// TIA Portal V15.1 export
// export: Created 2024-05-17T05:38:49.0670589Z, ExportSetting WithDefaults, DisplayName Totally Integrated Automation Portal, DisplayVersion V15.1 Update 5, DisplayName TIA Portal Openness, DisplayVersion V15.1 Update 5, DisplayName SINAMICS Startdrive Advanced, DisplayVersion V15.1, DisplayName G130, G150, S120, S150, SINAMICS MV, S210, DisplayVersion V15.1, DisplayName G110M, G120, G120C, G120D, G120P, DisplayVersion V15.1, DisplayName STEP 7 Professional, DisplayVersion V15.1 Update 5, DisplayName STEP 7 Safety, DisplayVersion V15.1, DisplayName WinCC Professional, DisplayVersion V15.1 Update 5, DisplayName SIMATIC Visualization Architect, DisplayVersion V15.1
FUNCTION_BLOCK "LGBExtCross2W2S-MoviFitFCPN"   // FB6653, FBD
TITLE = LGBExtCross2W2S-MoviFitFCPN
{ S7_Optimized_Access := 'TRUE' }
AUTHOR : ENGIE
FAMILY : Actuator
VERSION : 0.1
// stored: AutoNumber false, IsIECCheckEnabled false, IsRetainMemResEnabled false, MemoryReserve 100, SetENOAutomatically False, UDAEnableTagReadback false
   VAR_INPUT
      I_MotorProtection { ExternalAccessible := 'False'; ExternalVisible := 'False'; ExternalWritable := 'False'} : Bool;   // Motor protection
      I_BeltControlLeftDet { ExternalAccessible := 'False'; ExternalVisible := 'False'; ExternalWritable := 'False'} : Bool;   // Sensor Belt Control CrossConv left
      I_BeltControlRightDet { ExternalAccessible := 'False'; ExternalVisible := 'False'; ExternalWritable := 'False'} : Bool;   // Sensor Belt Control CrossConv right
      I_AlarmResetPB { ExternalAccessible := 'False'; ExternalVisible := 'False'; ExternalWritable := 'False'} : Bool;   // Alarm Reset Pushbutton is Activated
      I_SafetyStatusWord { ExternalAccessible := 'False'; ExternalVisible := 'False'; ExternalWritable := 'False'} : Word;   // Safety status word
      I_SafetyControlWord { ExternalAccessible := 'False'; ExternalVisible := 'False'; ExternalWritable := 'False'} : Word;   // Safety control word
      I_SafetyOk { ExternalAccessible := 'False'; ExternalVisible := 'False'; ExternalWritable := 'False'} : Bool;   // Safety ok
      I_MotionStopOk { ExternalAccessible := 'False'; ExternalVisible := 'False'; ExternalWritable := 'False'} : Bool;   // Safety Ok / The motion stop is Ok
      I_LSpdSetMotorCmd { ExternalAccessible := 'False'; ExternalVisible := 'False'; ExternalWritable := 'False'} : Bool;   // Low speed Set Command from function after interlock
      I_HSpdSetMotorCmd { ExternalAccessible := 'False'; ExternalVisible := 'False'; ExternalWritable := 'False'} : Bool;   // High Speed Set Command from function after Interlock
      I_LSpdResMotorCmd { ExternalAccessible := 'False'; ExternalVisible := 'False'; ExternalWritable := 'False'} : Bool;   // Low speed Reset Command from function after interlock
      I_HSpdResMotorCmd { ExternalAccessible := 'False'; ExternalVisible := 'False'; ExternalWritable := 'False'} : Bool;   // High speed Reset Command from function after Interlock
      I_LowSpeed { ExternalAccessible := 'False'; ExternalVisible := 'False'; ExternalWritable := 'False'} : Real;   // Low speed value 0-100%
      I_HighSpeed { ExternalAccessible := 'False'; ExternalVisible := 'False'; ExternalWritable := 'False'} : Real;   // High speed value 0-100%
      I_ReleaseBrake { ExternalAccessible := 'False'; ExternalVisible := 'False'; ExternalWritable := 'False'} : Bool;   // Release brake
   END_VAR
   VAR_OUTPUT
      O_ReleaseBrake { ExternalAccessible := 'False'; ExternalVisible := 'False'; ExternalWritable := 'False'} : Bool;   // Release the brake of the Motor
      O_Active { ExternalAccessible := 'False'; ExternalVisible := 'False'; ExternalWritable := 'False'} : Bool;   // Motor loop Active
      O_AlarmABCondition { ExternalAccessible := 'False'; ExternalVisible := 'False'; ExternalWritable := 'False'} : Bool;   // Alarm AB Condition
      O_AlarmA { ExternalAccessible := 'False'; ExternalVisible := 'False'; ExternalWritable := 'False'} : Bool;   // Alarm A
      O_AlarmB { ExternalAccessible := 'False'; ExternalVisible := 'False'; ExternalWritable := 'False'} : Bool;   // Alarm B
      O_AlarmC { ExternalAccessible := 'False'; ExternalVisible := 'False'; ExternalWritable := 'False'} : Bool;   // Alarm C
      O_AlarmD { ExternalAccessible := 'False'; ExternalVisible := 'False'; ExternalWritable := 'False'} : Bool;   // Alarm D
      H_AlarmDWord { ExternalAccessible := 'False'; ExternalVisible := 'False'; ExternalWritable := 'False'} : DWord;   // Alarm Word
   END_VAR
   VAR_IN_OUT
      IO_Modes : "Modes";   // Modes
      H_HMI : "H_HMI";
      "H_GBExtCross2W2S-MoviFitFCPN" : "H_GBExtCross2W2S-MoviFitFCPN";   // HMI UDT
      C_Config : "ExtCrossConfig";   // Config
   END_VAR
   VAR
      AA_MotorProtector { ExternalAccessible := 'False'; ExternalVisible := 'False'; ExternalWritable := 'False'} : Bool;   // Motorprotection Tripped / Motor Protection Tripped
      AA_SafetySwitch { ExternalAccessible := 'False'; ExternalVisible := 'False'; ExternalWritable := 'False'} : Bool;   // Safety Switch Not Ok
      AA_NoBusControl { ExternalAccessible := 'False'; ExternalVisible := 'False'; ExternalWritable := 'False'} : Bool;   // Bus control inactive
      AB_STO { ExternalAccessible := 'False'; ExternalVisible := 'False'; ExternalWritable := 'False'} : Bool;   // Safety Switch Not Ok / Safety output to drive is active but no response from drive that the safety is ok (STO)
      AB_BeltControlLeftDet { ExternalAccessible := 'False'; ExternalVisible := 'False'; ExternalWritable := 'False'} : Bool;   // Belt Check Cross Conveyor Left Side
      AB_BeltControlRightDet { ExternalAccessible := 'False'; ExternalVisible := 'False'; ExternalWritable := 'False'} : Bool;   // Belt Check Cross Conveyor Right Side
      AB_Alarm { ExternalAccessible := 'False'; ExternalVisible := 'False'; ExternalWritable := 'False'} : Bool;   // Frequency Control
      AD_Warning { ExternalAccessible := 'False'; ExternalVisible := 'False'; ExternalWritable := 'False'} : Bool;   // Frequency Control
      AD_MotionStop { ExternalAccessible := 'False'; ExternalVisible := 'False'; ExternalWritable := 'False'} : Bool;   // Motion Stop
      SafetyOk { ExternalAccessible := 'False'; ExternalVisible := 'False'; ExternalWritable := 'False'} : Bool;   // Safety Ok
      ParameterSet { ExternalAccessible := 'False'; ExternalVisible := 'False'; ExternalWritable := 'False'} : Bool;   // Active parameter set
      SetFrequency { ExternalAccessible := 'False'; ExternalVisible := 'False'; ExternalWritable := 'False'} : Real;   // Set frequency dependant on config
      ResFrequency { ExternalAccessible := 'False'; ExternalVisible := 'False'; ExternalWritable := 'False'} : Real;   // Reset frequency dependant on config
      MotorProtectionAlarmABCond { ExternalAccessible := 'False'; ExternalVisible := 'False'; ExternalWritable := 'False'} : Bool;   // Motor protection alarm condition
      SafetySwitchAlarmABCond { ExternalAccessible := 'False'; ExternalVisible := 'False'; ExternalWritable := 'False'} : Bool;   // Safety Switch alarm condition
      DriveFaultAlarm { ExternalAccessible := 'False'; ExternalVisible := 'False'; ExternalWritable := 'False'} : Bool;   // Drive fault alarm
      DriveFaultAlarmABCond { ExternalAccessible := 'False'; ExternalVisible := 'False'; ExternalWritable := 'False'} : Bool;   // Drive fault alarm condition
      STOAlarmABCond { ExternalAccessible := 'False'; ExternalVisible := 'False'; ExternalWritable := 'False'} : Bool;   // Drive fault alarm condition / STO feedback fault alarm condition
      EnableAlarmHWSR { ExternalAccessible := 'False'; ExternalVisible := 'False'; ExternalWritable := 'False'} : Bool;   // Enable Alarms from the hardware
      EnableAlarmHW { ExternalAccessible := 'False'; ExternalVisible := 'False'; ExternalWritable := 'False'} : Bool;   // Enable Alarms from the hardware
      Start { ExternalAccessible := 'False'; ExternalVisible := 'False'; ExternalWritable := 'False'} : Bool;   // Start command to drive
      SetpointSpeed { ExternalAccessible := 'False'; ExternalVisible := 'False'; ExternalWritable := 'False'} : Real;   // Setpoint speed
      SetpointSpeedCalc { ExternalAccessible := 'False'; ExternalVisible := 'False'; ExternalWritable := 'False'} : Real;   // Setpoint speed to drive / Setpoint speed
      OutputStageEnabled { ExternalAccessible := 'False'; ExternalVisible := 'False'; ExternalWritable := 'False'} : Bool;   // Inverter output stage is enabled
      MaintenanceSwitch { ExternalAccessible := 'False'; ExternalVisible := 'False'; ExternalWritable := 'False'} : Bool;   // Maintenance switch activated (1=mains OFF)
      PODataEnabled { ExternalAccessible := 'False'; ExternalVisible := 'False'; ExternalWritable := 'False'} : Bool;   // Process data is enabled (1 = Drive can be controlled via fieldbus)
      PODataDisabled { ExternalAccessible := 'False'; ExternalVisible := 'False'; ExternalWritable := 'False'} : Bool;   // Process data is enabled (1 = Drive can be controlled via fieldbus)
      Fault { ExternalAccessible := 'False'; ExternalVisible := 'False'; ExternalWritable := 'False'} : Bool;   // Fault present
      Brake { ExternalAccessible := 'False'; ExternalVisible := 'False'; ExternalWritable := 'False'} : Bool;   // Brake status
      ActorVoltageOverloadDO00 { ExternalAccessible := 'False'; ExternalVisible := 'False'; ExternalWritable := 'False'} : Bool;   // Short circuit / overload of the actuator voltage for digital output DO00
      ActorVoltageOverloadDO01 { ExternalAccessible := 'False'; ExternalVisible := 'False'; ExternalWritable := 'False'} : Bool;   // Short circuit / overload of the actuator voltage for digital output DO01
      ActorVoltageOverloadDO02 { ExternalAccessible := 'False'; ExternalVisible := 'False'; ExternalWritable := 'False'} : Bool;   // Short circuit / overload of the actuator voltage for digital output DO02
      ActorVoltageOverloadDO03 { ExternalAccessible := 'False'; ExternalVisible := 'False'; ExternalWritable := 'False'} : Bool;   // Short circuit / overload of the actuator voltage for digital output DO03
      SensorVoltageOverloadGroup1 { ExternalAccessible := 'False'; ExternalVisible := 'False'; ExternalWritable := 'False'} : Bool;   // Short circuit / overload of the sensor suuply group 1 (VO24-I)
      SensorVoltageOverloadGroup2 { ExternalAccessible := 'False'; ExternalVisible := 'False'; ExternalWritable := 'False'} : Bool;   // Short circuit / overload of the sensor suuply group 2 (VO24-I)
      SensorVoltageOverloadGroup3 { ExternalAccessible := 'False'; ExternalVisible := 'False'; ExternalWritable := 'False'} : Bool;   // Short circuit / overload of the sensor suuply group 3 (VO24-I)
      SensorVoltageOverloadGroup4 { ExternalAccessible := 'False'; ExternalVisible := 'False'; ExternalWritable := 'False'} : Bool;   // Short circuit / overload of the sensor suuply group 4 (VO24-I)
      "Undervoltage24V-S" { ExternalAccessible := 'False'; ExternalVisible := 'False'; ExternalWritable := 'False'} : Bool;   // Value falls below the power limit for the actuator voltage DO00-03
      "InverterVoltageNotApplied24V-P" { ExternalAccessible := 'False'; ExternalVisible := 'False'; ExternalWritable := 'False'} : Bool;   // Presence of 24V_P for integrated inverter (FC) or external MOVIMOT (1=24V_P not present)
      MOVIFITSystemFault { ExternalAccessible := 'False'; ExternalVisible := 'False'; ExternalWritable := 'False'} : Bool;   // MOVIFIT system fault
      DriveReady { ExternalAccessible := 'False'; ExternalVisible := 'False'; ExternalWritable := 'False'} : Bool;   // Motor Loop Active / Drive ready
      BeltControlLeftAlarmABCondition { ExternalAccessible := 'False'; ExternalVisible := 'False'; ExternalWritable := 'False'} : Bool;   // Belt Control AB Condition
      BeltControlRightAlarmABCondition { ExternalAccessible := 'False'; ExternalVisible := 'False'; ExternalWritable := 'False'} : Bool;   // Belt Control AB Condition
      BeltPulseCountLeft { ExternalAccessible := 'False'; ExternalVisible := 'False'; ExternalWritable := 'False'} : DInt;   // Temp
      BeltPulseCountRight { ExternalAccessible := 'False'; ExternalVisible := 'False'; ExternalWritable := 'False'} : DInt;   // Temp
      BeltPosEdgeLeft1 { ExternalAccessible := 'False'; ExternalVisible := 'False'; ExternalWritable := 'False'} : Bool;   // Pos Edge
      BeltPosEdgeLeft2 { ExternalAccessible := 'False'; ExternalVisible := 'False'; ExternalWritable := 'False'} : Bool;   // Pos Edge
      BeltPosEdgeRight1 { ExternalAccessible := 'False'; ExternalVisible := 'False'; ExternalWritable := 'False'} : Bool;   // Pos Edge
      BeltPosEdgeRight2 { ExternalAccessible := 'False'; ExternalVisible := 'False'; ExternalWritable := 'False'} : Bool;   // Pos Edge
      InitBeltCounterLeft { ExternalAccessible := 'False'; ExternalVisible := 'False'; ExternalWritable := 'False'} : Bool;   // Init
      InitBeltCounterRight { ExternalAccessible := 'False'; ExternalVisible := 'False'; ExternalWritable := 'False'} : Bool;   // Init
      AlarmA { ExternalAccessible := 'False'; ExternalVisible := 'False'; ExternalWritable := 'False'} : Bool;   // Alarm A
      AlarmB { ExternalAccessible := 'False'; ExternalVisible := 'False'; ExternalWritable := 'False'} : Bool;   // Alarm B
      AlarmC { ExternalAccessible := 'False'; ExternalVisible := 'False'; ExternalWritable := 'False'} : Bool;   // Alarm C
      AlarmD { ExternalAccessible := 'False'; ExternalVisible := 'False'; ExternalWritable := 'False'} : Bool;   // Alarm D
      Ramp { ExternalAccessible := 'False'; ExternalVisible := 'False'; ExternalWritable := 'False'} : DInt;   // Ramp
      RampToDrive { ExternalAccessible := 'False'; ExternalVisible := 'False'; ExternalWritable := 'False'} : Time;   // Calculated Ramp send in miliseconds
      _BeltControlRight { ExternalAccessible := 'False'; ExternalVisible := 'False'; ExternalWritable := 'False'} : "L1AlarmMultiIn";   // FB
      _BeltControlLeft { ExternalAccessible := 'False'; ExternalVisible := 'False'; ExternalWritable := 'False'} : "L1AlarmMultiIn";   // FB
      _InitBeltCntLeft { ExternalAccessible := 'False'; ExternalVisible := 'False'; ExternalWritable := 'False'} : "LChangeOfState";   // FB
      _InitBeltCntRight { ExternalAccessible := 'False'; ExternalVisible := 'False'; ExternalWritable := 'False'} : "LChangeOfState";   // FB
      _MoviFitPN { ExternalAccessible := 'False'; ExternalVisible := 'False'; ExternalWritable := 'False'} : "LGBSEW-MoviFitFCPN";   // FB / SEW MOVIFIT FC
      _MotorProtection { ExternalAccessible := 'False'; ExternalVisible := 'False'; ExternalWritable := 'False'} : "L1AlarmMultiIn";   // FB
      _SafetySwitch { ExternalAccessible := 'False'; ExternalVisible := 'False'; ExternalWritable := 'False'} : "L1AlarmMultiIn";   // FB
      _DriveFault { ExternalAccessible := 'False'; ExternalVisible := 'False'; ExternalWritable := 'False'} : "L1AlarmMultiIn";   // FB
      _STO { ExternalAccessible := 'False'; ExternalVisible := 'False'; ExternalWritable := 'False'} : "L1AlarmMultiIn";   // FB
      _MotionStop { ExternalAccessible := 'False'; ExternalVisible := 'False'; ExternalWritable := 'False'} : "L1AlarmMultiIn";   // FB
      T_STOAlarm { ExternalAccessible := 'False'; ExternalVisible := 'False'; ExternalWritable := 'False'} : TON_TIME;   // Timer
      T_Reboot { ExternalAccessible := 'False'; ExternalVisible := 'False'; ExternalWritable := 'False'} : TON_TIME;   // Timer
   END_VAR
   VAR_TEMP   // added for the SCL form of the ladder/FBD networks
      _w1 : Bool;
      _w2 : Bool;
      _w3 : Bool;
      _w4 : Bool;
   END_VAR
BEGIN

NETWORK
TITLE = **** 1 - Inputs **** Init Belt Control Set And Reset Direction
// Init Belt Control Set And Reset Direction
      CALL  #_InitBeltCntLeft
      ( I_In     := #I_BeltControlLeftDet,
        O_OutPut := #InitBeltCounterLeft
      );
      NOP   0;

      CALL  #_InitBeltCntRight
      ( I_In     := #I_BeltControlRightDet,
        O_OutPut := #InitBeltCounterRight
      );
      NOP   0;

      A(;
      O     #InitBeltCounterLeft;
      O;
      A     #IO_Modes.LMode.ManualMode;
      A     #IO_Modes.LMode.AlarmResetPB;
      );
      JCN   NCSet;
      L     0;
      T     #BeltPulseCountLeft;
NCSet:NOP   0;

      A(;
      O     #InitBeltCounterRight;
      O;
      A     #IO_Modes.LMode.ManualMode;
      A     #IO_Modes.LMode.AlarmResetPB;
      );
      JCN   NCReset;
      L     0;
      T     #BeltPulseCountRight;
NCReset:NOP   0;


REGION Network 2: **** 1 - Inputs **** Safety Ok
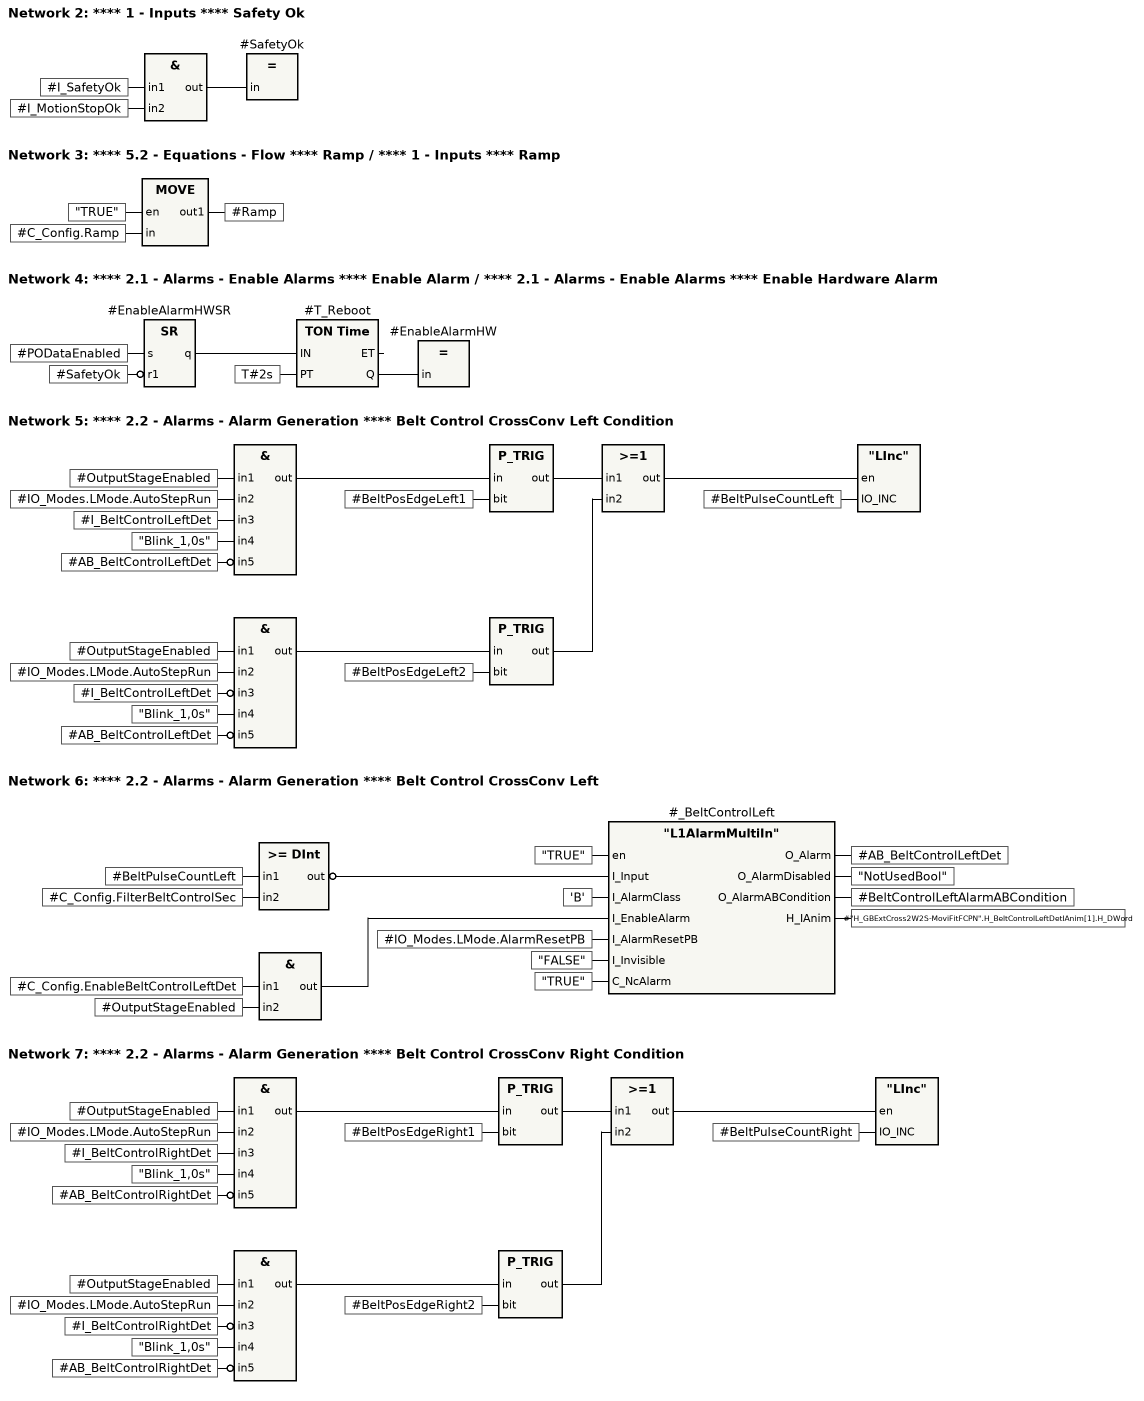
   #SafetyOk := #I_SafetyOk AND #I_MotionStopOk;
END_REGION

REGION Network 3: **** 5.2 - Equations - Flow **** Ramp / **** 1 - Inputs **** Ramp
   IF "TRUE" THEN #Ramp := #C_Config.Ramp; END_IF;
END_REGION

REGION Network 4: **** 2.1 - Alarms - Enable Alarms **** Enable Alarm / **** 2.1 - Alarms - Enable Alarms **** Enable Hardware Alarm
   // Enable Alarm / Enable Hardware Alarm
   IF #PODataEnabled THEN
       #EnableAlarmHWSR := TRUE;   // SR flip-flop
   END_IF;
   IF NOT #SafetyOk THEN #EnableAlarmHWSR := FALSE; END_IF;
   #T_Reboot(IN := #EnableAlarmHWSR, PT := T#2s);   // TON
   #EnableAlarmHW := #T_Reboot.Q;
END_REGION

REGION Network 5: **** 2.2 - Alarms - Alarm Generation **** Belt Control CrossConv Left Condition
   // Belt Control CrossConv Set Condition
   #_w1 := #OutputStageEnabled AND #IO_Modes.LMode.AutoStepRun AND #I_BeltControlLeftDet AND "Blink_1,0s" AND NOT #AB_BeltControlLeftDet;
   #_w2 := #_w1 AND NOT #BeltPosEdgeLeft1;   // rising edge
   #BeltPosEdgeLeft1 := #_w1;
   #_w3 := #OutputStageEnabled AND #IO_Modes.LMode.AutoStepRun AND NOT #I_BeltControlLeftDet AND "Blink_1,0s" AND NOT #AB_BeltControlLeftDet;
   #_w4 := #_w3 AND NOT #BeltPosEdgeLeft2;   // rising edge
   #BeltPosEdgeLeft2 := #_w3;
   IF #_w2 OR #_w4 THEN "LInc"(IO_INC := #BeltPulseCountLeft); END_IF;
END_REGION

REGION Network 6: **** 2.2 - Alarms - Alarm Generation **** Belt Control CrossConv Left
   // Belt Control CrossConv Set
   IF "TRUE" THEN
       #_BeltControlLeft(I_Input := NOT (#BeltPulseCountLeft >= #C_Config.FilterBeltControlSec),   // "L1AlarmMultiIn"
                         I_AlarmClass := 'B',
                         I_EnableAlarm := #C_Config.EnableBeltControlLeftDet AND #OutputStageEnabled,
                         I_AlarmResetPB := #IO_Modes.LMode.AlarmResetPB,
                         I_Invisible := "FALSE",
                         C_NcAlarm := "TRUE",
                         O_Alarm => #AB_BeltControlLeftDet,
                         O_AlarmDisabled => "NotUsedBool",
                         O_AlarmABCondition => #BeltControlLeftAlarmABCondition,
                         H_IAnim => #"H_GBExtCross2W2S-MoviFitFCPN".H_BeltControlLeftDetIAnim[1].H_DWord);
   END_IF;
END_REGION

REGION Network 7: **** 2.2 - Alarms - Alarm Generation **** Belt Control CrossConv Right Condition
   // Belt Control CrossConv Set Condition
   #_w1 := #OutputStageEnabled AND #IO_Modes.LMode.AutoStepRun AND #I_BeltControlRightDet AND "Blink_1,0s" AND NOT #AB_BeltControlRightDet;
   #_w2 := #_w1 AND NOT #BeltPosEdgeRight1;   // rising edge
   #BeltPosEdgeRight1 := #_w1;
   #_w3 := #OutputStageEnabled AND #IO_Modes.LMode.AutoStepRun AND NOT #I_BeltControlRightDet AND "Blink_1,0s" AND NOT #AB_BeltControlRightDet;
   #_w4 := #_w3 AND NOT #BeltPosEdgeRight2;   // rising edge
   #BeltPosEdgeRight2 := #_w3;
   IF #_w2 OR #_w4 THEN "LInc"(IO_INC := #BeltPulseCountRight); END_IF;
END_REGION

REGION Network 8: **** 2.2 - Alarms - Alarm Generation **** Belt Control CrossConv Right
   // Belt Control CrossConv Set
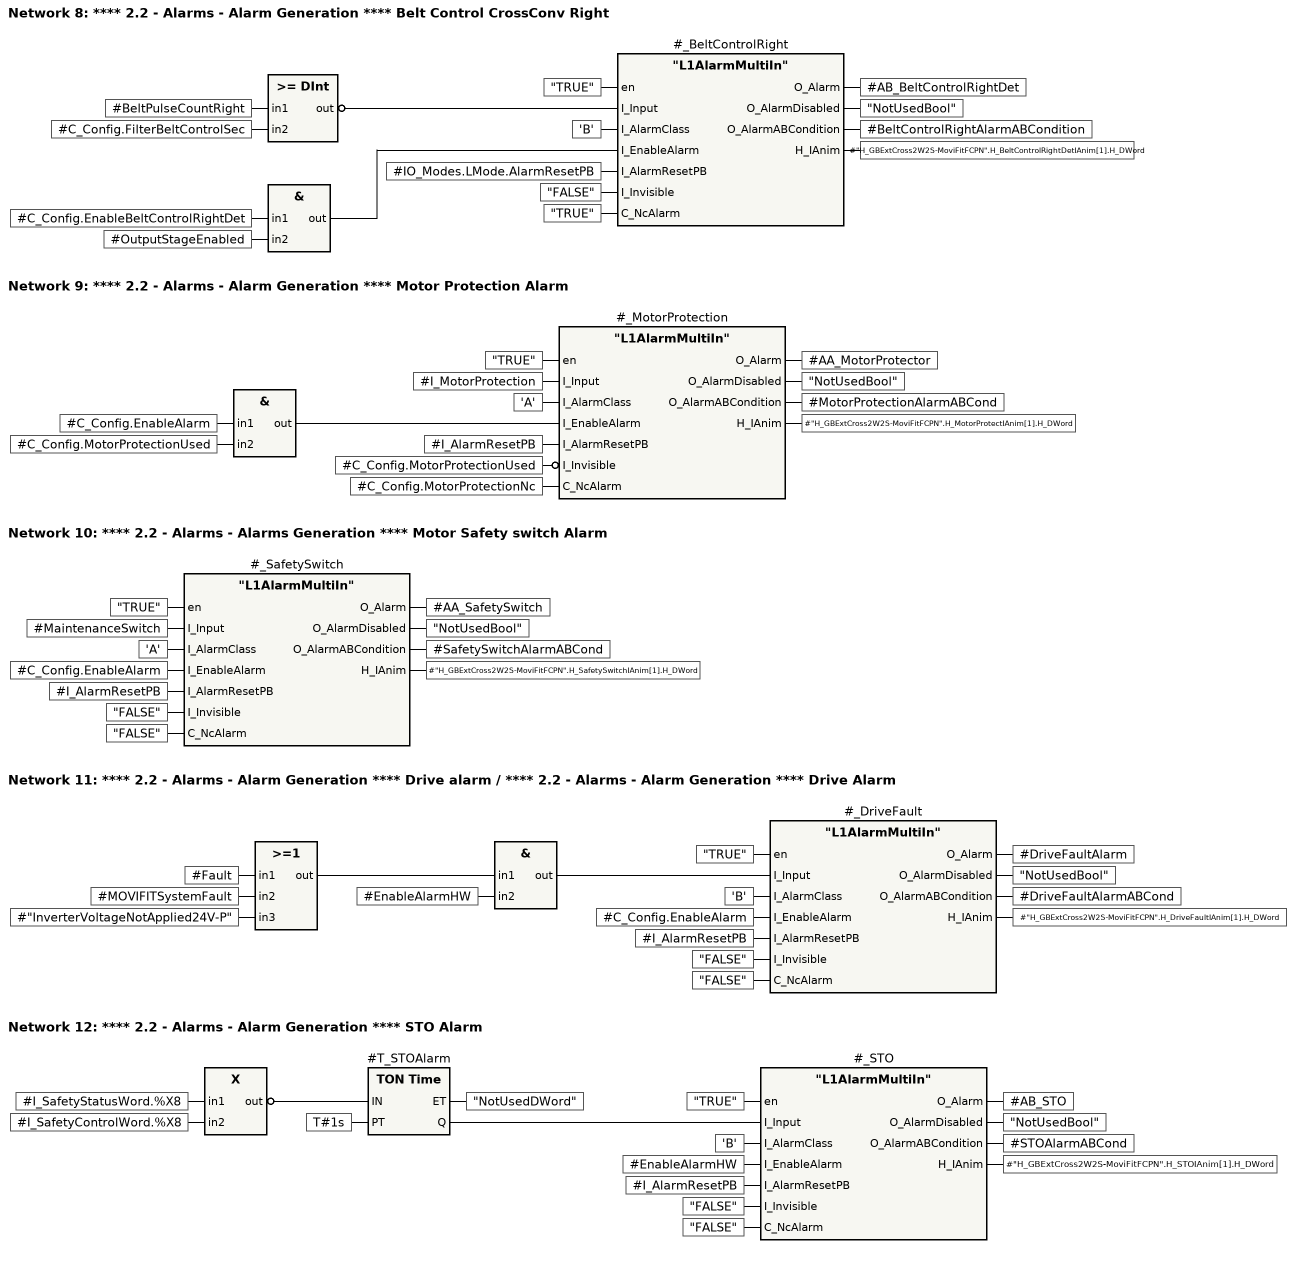
   IF "TRUE" THEN
       #_BeltControlRight(I_Input := NOT (#BeltPulseCountRight >= #C_Config.FilterBeltControlSec),   // "L1AlarmMultiIn"
                          I_AlarmClass := 'B',
                          I_EnableAlarm := #C_Config.EnableBeltControlRightDet AND #OutputStageEnabled,
                          I_AlarmResetPB := #IO_Modes.LMode.AlarmResetPB,
                          I_Invisible := "FALSE",
                          C_NcAlarm := "TRUE",
                          O_Alarm => #AB_BeltControlRightDet,
                          O_AlarmDisabled => "NotUsedBool",
                          O_AlarmABCondition => #BeltControlRightAlarmABCondition,
                          H_IAnim => #"H_GBExtCross2W2S-MoviFitFCPN".H_BeltControlRightDetIAnim[1].H_DWord);
   END_IF;
END_REGION

REGION Network 9: **** 2.2 - Alarms - Alarm Generation **** Motor Protection Alarm
   // Motor Protection Alarm
   IF "TRUE" THEN
       #_MotorProtection(I_Input := #I_MotorProtection,   // "L1AlarmMultiIn"
                         I_AlarmClass := 'A',
                         I_EnableAlarm := #C_Config.EnableAlarm AND #C_Config.MotorProtectionUsed,
                         I_AlarmResetPB := #I_AlarmResetPB,
                         I_Invisible := NOT #C_Config.MotorProtectionUsed,
                         C_NcAlarm := #C_Config.MotorProtectionNc,
                         O_Alarm => #AA_MotorProtector,
                         O_AlarmDisabled => "NotUsedBool",
                         O_AlarmABCondition => #MotorProtectionAlarmABCond,
                         H_IAnim => #"H_GBExtCross2W2S-MoviFitFCPN".H_MotorProtectIAnim[1].H_DWord);
   END_IF;
END_REGION

REGION Network 10: **** 2.2 - Alarms - Alarms Generation **** Motor Safety switch Alarm
   // Motor Safety switch Alarm
   IF "TRUE" THEN
       #_SafetySwitch(I_Input := #MaintenanceSwitch,   // "L1AlarmMultiIn"
                      I_AlarmClass := 'A',
                      I_EnableAlarm := #C_Config.EnableAlarm,
                      I_AlarmResetPB := #I_AlarmResetPB,
                      I_Invisible := "FALSE",
                      C_NcAlarm := "FALSE",
                      O_Alarm => #AA_SafetySwitch,
                      O_AlarmDisabled => "NotUsedBool",
                      O_AlarmABCondition => #SafetySwitchAlarmABCond,
                      H_IAnim => #"H_GBExtCross2W2S-MoviFitFCPN".H_SafetySwitchIAnim[1].H_DWord);
   END_IF;
END_REGION

REGION Network 11: **** 2.2 - Alarms - Alarm Generation **** Drive alarm / **** 2.2 - Alarms - Alarm Generation **** Drive Alarm
   IF "TRUE" THEN
       #_DriveFault(I_Input := (#Fault OR #MOVIFITSystemFault OR #"InverterVoltageNotApplied24V-P") AND #EnableAlarmHW,   // "L1AlarmMultiIn"
                    I_AlarmClass := 'B',
                    I_EnableAlarm := #C_Config.EnableAlarm,
                    I_AlarmResetPB := #I_AlarmResetPB,
                    I_Invisible := "FALSE",
                    C_NcAlarm := "FALSE",
                    O_Alarm => #DriveFaultAlarm,
                    O_AlarmDisabled => "NotUsedBool",
                    O_AlarmABCondition => #DriveFaultAlarmABCond,
                    H_IAnim => #"H_GBExtCross2W2S-MoviFitFCPN".H_DriveFaultIAnim[1].H_DWord);
   END_IF;
END_REGION

REGION Network 12: **** 2.2 - Alarms - Alarm Generation **** STO Alarm
   #T_STOAlarm(IN := NOT (#I_SafetyStatusWord.%X8 XOR #I_SafetyControlWord.%X8),   // TON
               PT := T#1s,
               ET => "NotUsedDWord");
   IF "TRUE" THEN
       #_STO(I_Input := #T_STOAlarm.Q,   // "L1AlarmMultiIn"
             I_AlarmClass := 'B',
             I_EnableAlarm := #EnableAlarmHW,
             I_AlarmResetPB := #I_AlarmResetPB,
             I_Invisible := "FALSE",
             C_NcAlarm := "FALSE",
             O_Alarm => #AB_STO,
             O_AlarmDisabled => "NotUsedBool",
             O_AlarmABCondition => #STOAlarmABCond,
             H_IAnim => #"H_GBExtCross2W2S-MoviFitFCPN".H_STOIAnim[1].H_DWord);
   END_IF;
END_REGION

REGION Network 13: **** 2.2 - Alarms - Alarm Generation **** MotionStop Warning
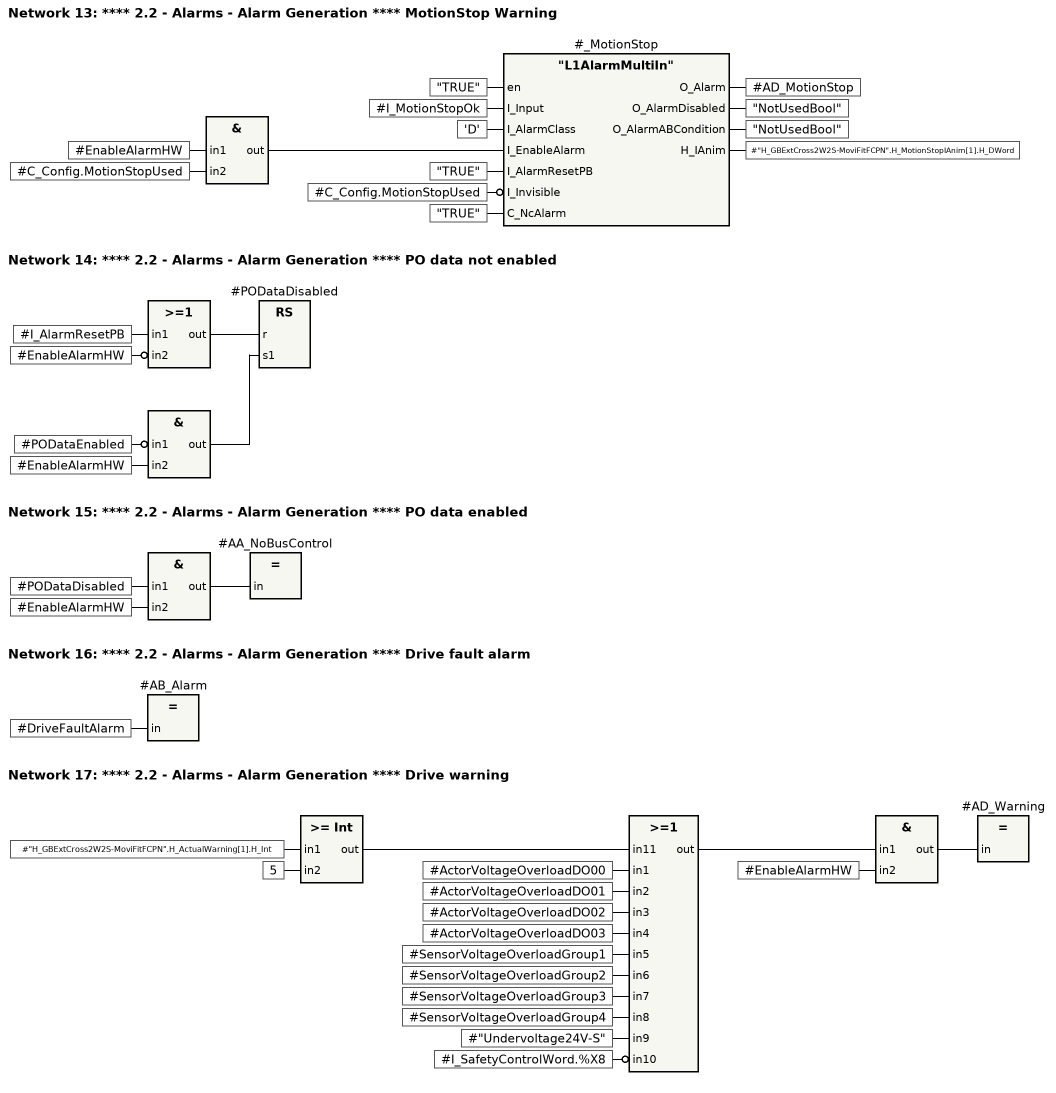
   IF "TRUE" THEN
       #_MotionStop(I_Input := #I_MotionStopOk,   // "L1AlarmMultiIn"
                    I_AlarmClass := 'D',
                    I_EnableAlarm := #EnableAlarmHW AND #C_Config.MotionStopUsed,
                    I_AlarmResetPB := "TRUE",
                    I_Invisible := NOT #C_Config.MotionStopUsed,
                    C_NcAlarm := "TRUE",
                    O_Alarm => #AD_MotionStop,
                    O_AlarmDisabled => "NotUsedBool",
                    O_AlarmABCondition => "NotUsedBool",
                    H_IAnim => #"H_GBExtCross2W2S-MoviFitFCPN".H_MotionStopIAnim[1].H_DWord);
   END_IF;
END_REGION

REGION Network 14: **** 2.2 - Alarms - Alarm Generation **** PO data not enabled
   IF #I_AlarmResetPB OR NOT #EnableAlarmHW THEN
       #PODataDisabled := FALSE;   // RS flip-flop
   END_IF;
   IF NOT #PODataEnabled AND #EnableAlarmHW THEN #PODataDisabled := TRUE; END_IF;
END_REGION

REGION Network 15: **** 2.2 - Alarms - Alarm Generation **** PO data enabled
   #AA_NoBusControl := #PODataDisabled AND #EnableAlarmHW;
END_REGION

REGION Network 16: **** 2.2 - Alarms - Alarm Generation **** Drive fault alarm
   // Drive fault
   #AB_Alarm := #DriveFaultAlarm;
END_REGION

REGION Network 17: **** 2.2 - Alarms - Alarm Generation **** Drive warning
   #AD_Warning := ((#"H_GBExtCross2W2S-MoviFitFCPN".H_ActualWarning[1].H_Int >= 5) OR #ActorVoltageOverloadDO00 OR #ActorVoltageOverloadDO01 OR #ActorVoltageOverloadDO02 OR #ActorVoltageOverloadDO03 OR #SensorVoltageOverloadGroup1 OR #SensorVoltageOverloadGroup2 OR #SensorVoltageOverloadGroup3 OR #SensorVoltageOverloadGroup4 OR #"Undervoltage24V-S" OR NOT #I_SafetyControlWord.%X8) AND #EnableAlarmHW;
END_REGION

REGION Network 18: **** 4.6 - Machine Status - Indication **** Icon Animation
   // Icon Animation
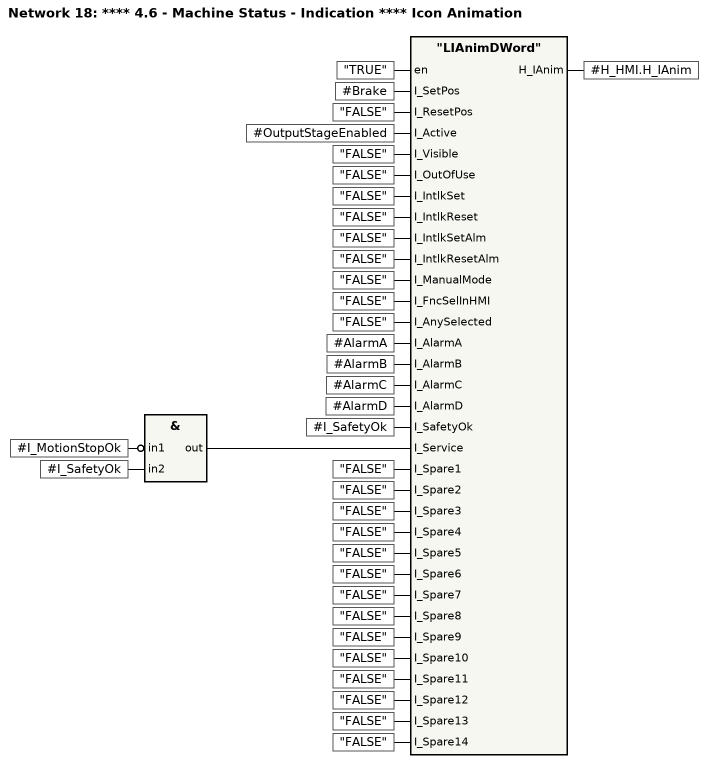
   IF "TRUE" THEN
       "LIAnimDWord"(I_SetPos := #Brake,
                     I_ResetPos := "FALSE",
                     I_Active := #OutputStageEnabled,
                     I_Visible := "FALSE",
                     I_OutOfUse := "FALSE",
                     I_IntlkSet := "FALSE",
                     I_IntlkReset := "FALSE",
                     I_IntlkSetAlm := "FALSE",
                     I_IntlkResetAlm := "FALSE",
                     I_ManualMode := "FALSE",
                     I_FncSelInHMI := "FALSE",
                     I_AnySelected := "FALSE",
                     I_AlarmA := #AlarmA,
                     I_AlarmB := #AlarmB,
                     I_AlarmC := #AlarmC,
                     I_AlarmD := #AlarmD,
                     I_SafetyOk := #I_SafetyOk,
                     I_Service := NOT #I_MotionStopOk AND #I_SafetyOk,
                     I_Spare1 := "FALSE",
                     I_Spare2 := "FALSE",
                     I_Spare3 := "FALSE",
                     I_Spare4 := "FALSE",
                     I_Spare5 := "FALSE",
                     I_Spare6 := "FALSE",
                     I_Spare7 := "FALSE",
                     I_Spare8 := "FALSE",
                     I_Spare9 := "FALSE",
                     I_Spare10 := "FALSE",
                     I_Spare11 := "FALSE",
                     I_Spare12 := "FALSE",
                     I_Spare13 := "FALSE",
                     I_Spare14 := "FALSE",
                     H_IAnim => #H_HMI.H_IAnim);
   END_IF;
END_REGION

REGION Network 19: **** 4.6 - Machine Status - Indication **** Animation
   // Animation
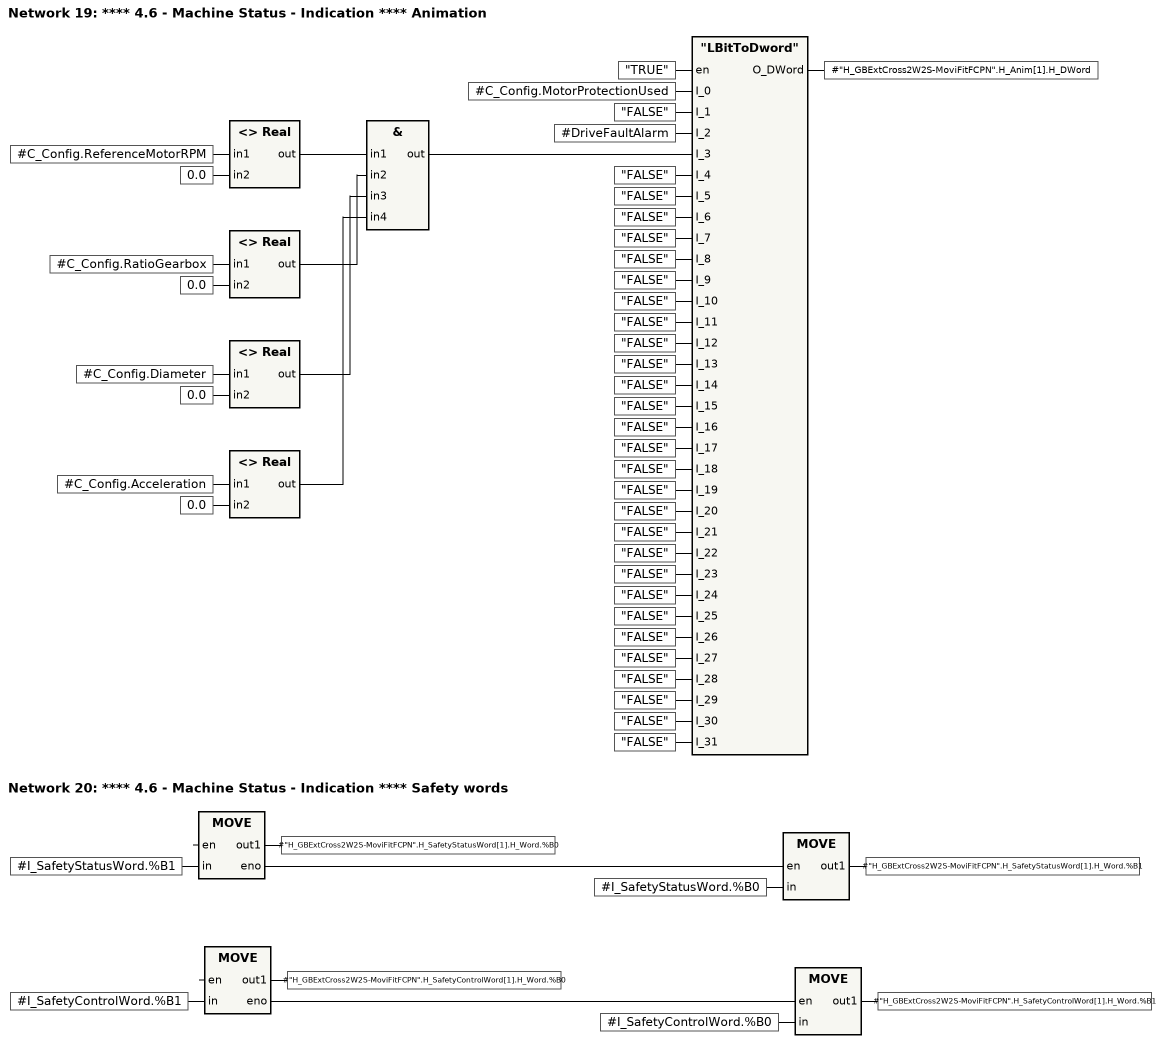
   IF "TRUE" THEN
       "LBitToDword"(I_0 := #C_Config.MotorProtectionUsed,
                     I_1 := "FALSE",
                     I_2 := #DriveFaultAlarm,
                     I_3 := (#C_Config.ReferenceMotorRPM <> 0.0) AND (#C_Config.RatioGearbox <> 0.0) AND (#C_Config.Diameter <> 0.0) AND (#C_Config.Acceleration <> 0.0),
                     I_4 := "FALSE",
                     I_5 := "FALSE",
                     I_6 := "FALSE",
                     I_7 := "FALSE",
                     I_8 := "FALSE",
                     I_9 := "FALSE",
                     I_10 := "FALSE",
                     I_11 := "FALSE",
                     I_12 := "FALSE",
                     I_13 := "FALSE",
                     I_14 := "FALSE",
                     I_15 := "FALSE",
                     I_16 := "FALSE",
                     I_17 := "FALSE",
                     I_18 := "FALSE",
                     I_19 := "FALSE",
                     I_20 := "FALSE",
                     I_21 := "FALSE",
                     I_22 := "FALSE",
                     I_23 := "FALSE",
                     I_24 := "FALSE",
                     I_25 := "FALSE",
                     I_26 := "FALSE",
                     I_27 := "FALSE",
                     I_28 := "FALSE",
                     I_29 := "FALSE",
                     I_30 := "FALSE",
                     I_31 := "FALSE",
                     O_DWord => #"H_GBExtCross2W2S-MoviFitFCPN".H_Anim[1].H_DWord);
   END_IF;
END_REGION

REGION Network 20: **** 4.6 - Machine Status - Indication **** Safety words
   // Animation
   #"H_GBExtCross2W2S-MoviFitFCPN".H_SafetyStatusWord[1].H_Word.%B0 := #I_SafetyStatusWord.%B1;
   #"H_GBExtCross2W2S-MoviFitFCPN".H_SafetyStatusWord[1].H_Word.%B1 := #I_SafetyStatusWord.%B0;
   #"H_GBExtCross2W2S-MoviFitFCPN".H_SafetyControlWord[1].H_Word.%B0 := #I_SafetyControlWord.%B1;
   #"H_GBExtCross2W2S-MoviFitFCPN".H_SafetyControlWord[1].H_Word.%B1 := #I_SafetyControlWord.%B0;
END_REGION

REGION Network 21: **** 5.2 - Equations - Flow **** Reverse Frequency
   // Reverse frequency dependant on config
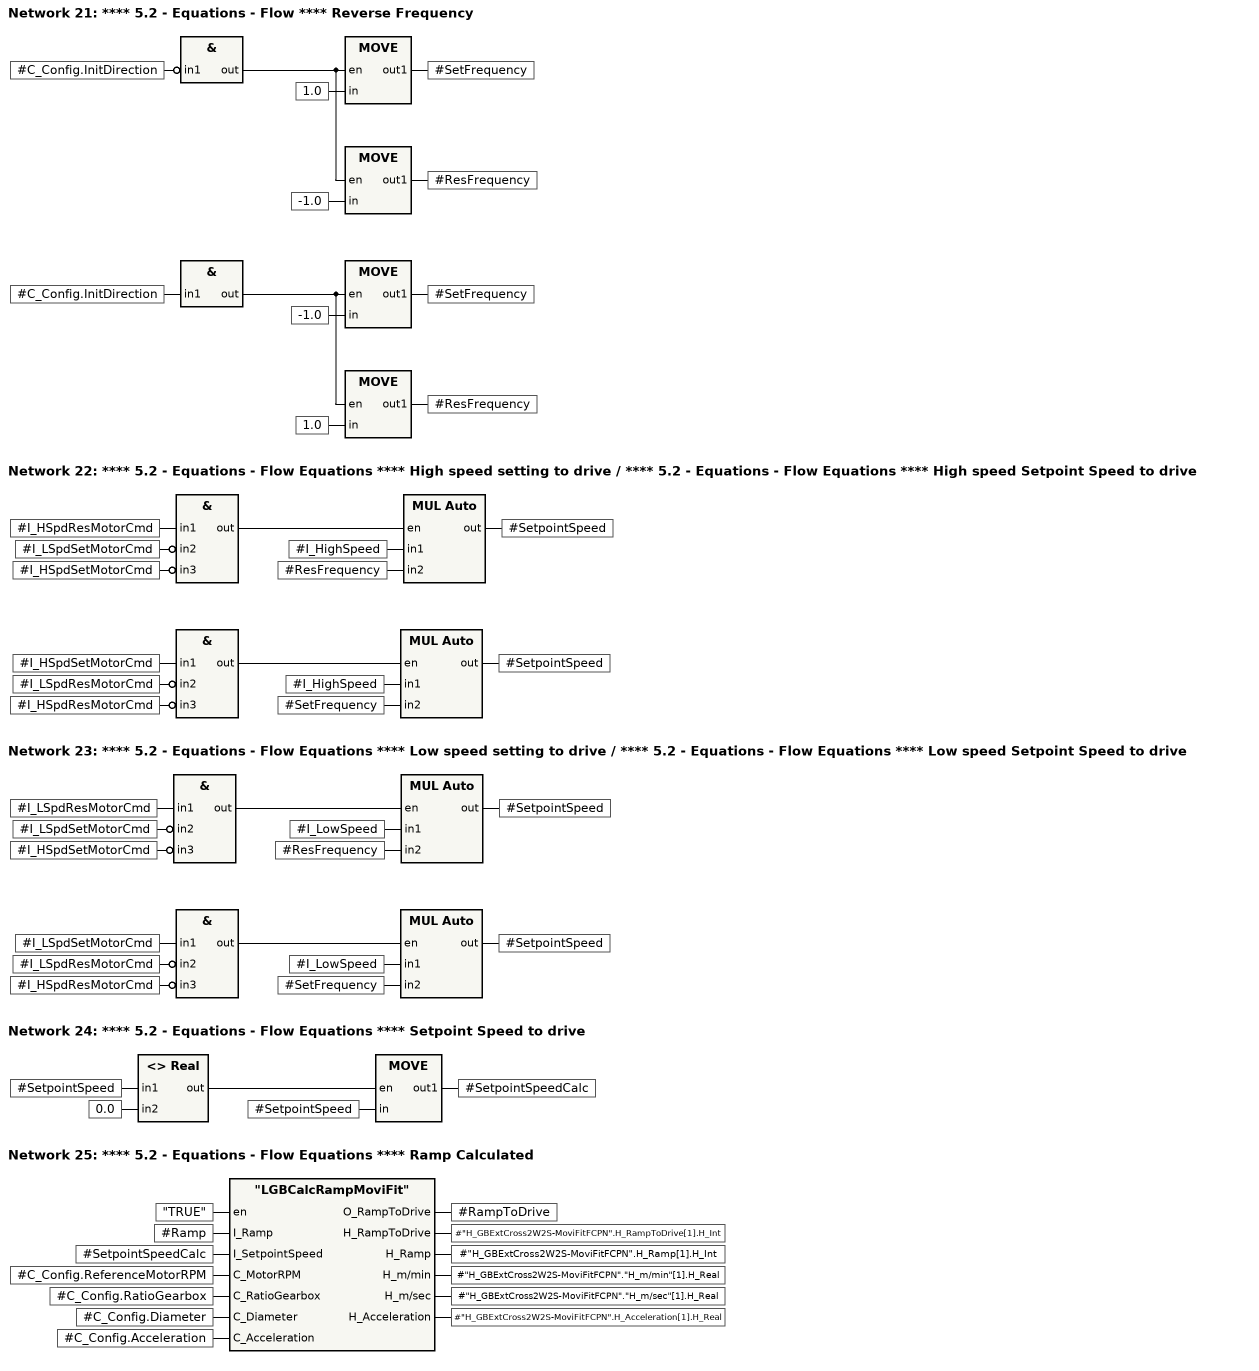
   IF NOT #C_Config.InitDirection THEN
       #SetFrequency := 1.0;
       #ResFrequency := -1.0;
   END_IF;
   IF #C_Config.InitDirection THEN
       #SetFrequency := -1.0;
       #ResFrequency := 1.0;
   END_IF;
END_REGION

REGION Network 22: **** 5.2 - Equations - Flow Equations **** High speed setting to drive / **** 5.2 - Equations - Flow Equations **** High speed Setpoint Speed to drive
   // Select high speed
   IF #I_HSpdResMotorCmd AND NOT #I_LSpdSetMotorCmd AND NOT #I_HSpdSetMotorCmd THEN
       #SetpointSpeed := #I_HighSpeed * #ResFrequency;
   END_IF;
   IF #I_HSpdSetMotorCmd AND NOT #I_LSpdResMotorCmd AND NOT #I_HSpdResMotorCmd THEN
       #SetpointSpeed := #I_HighSpeed * #SetFrequency;   // If multiple commands are active then set direction has prioritry over reset direction and Slow speed has priority over high speed. (dependant on the order of programming)
   END_IF;
END_REGION

REGION Network 23: **** 5.2 - Equations - Flow Equations **** Low speed setting to drive / **** 5.2 - Equations - Flow Equations **** Low speed Setpoint Speed to drive
   IF #I_LSpdResMotorCmd AND NOT #I_LSpdSetMotorCmd AND NOT #I_HSpdSetMotorCmd THEN
       #SetpointSpeed := #I_LowSpeed * #ResFrequency;
   END_IF;
   IF #I_LSpdSetMotorCmd AND NOT #I_LSpdResMotorCmd AND NOT #I_HSpdResMotorCmd THEN
       #SetpointSpeed := #I_LowSpeed * #SetFrequency;   // If multiple commands are active then set direction has prioritry over reset direction and Slow speed has priority over high speed. (dependant on the order of programming)
   END_IF;
END_REGION

REGION Network 24: **** 5.2 - Equations - Flow Equations **** Setpoint Speed to drive
   IF #SetpointSpeed <> 0.0 THEN #SetpointSpeedCalc := #SetpointSpeed; END_IF;
END_REGION

REGION Network 25: **** 5.2 - Equations - Flow Equations **** Ramp Calculated
   IF "TRUE" THEN
       "LGBCalcRampMoviFit"(I_Ramp := #Ramp,
                            I_SetpointSpeed := #SetpointSpeedCalc,
                            C_MotorRPM := #C_Config.ReferenceMotorRPM,
                            C_RatioGearbox := #C_Config.RatioGearbox,
                            C_Diameter := #C_Config.Diameter,
                            C_Acceleration := #C_Config.Acceleration,
                            O_RampToDrive => #RampToDrive,
                            H_RampToDrive => #"H_GBExtCross2W2S-MoviFitFCPN".H_RampToDrive[1].H_Int,
                            H_Ramp => #"H_GBExtCross2W2S-MoviFitFCPN".H_Ramp[1].H_Int,
                            "H_m/min" => #"H_GBExtCross2W2S-MoviFitFCPN"."H_m/min"[1].H_Real,
                            "H_m/sec" => #"H_GBExtCross2W2S-MoviFitFCPN"."H_m/sec"[1].H_Real,
                            H_Acceleration => #"H_GBExtCross2W2S-MoviFitFCPN".H_Acceleration[1].H_Real);
   END_IF;
END_REGION

REGION Network 26: **** 5.2 - Equations - Flow Equations **** Start command to drive
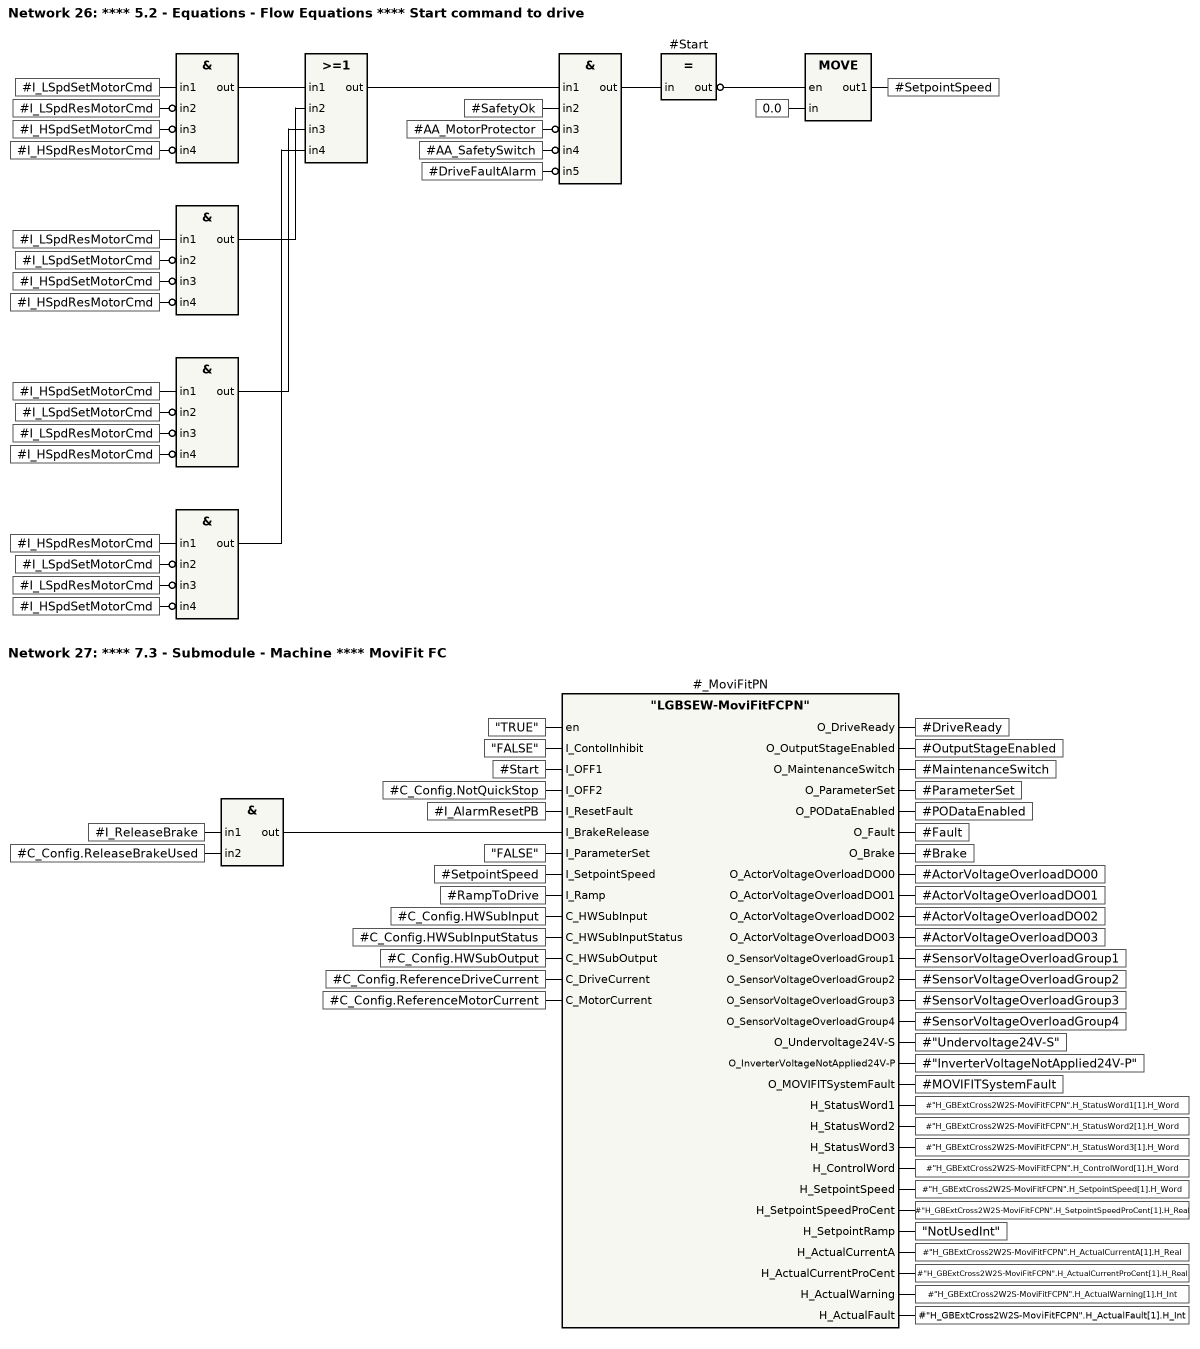
   #_w1 := ((#I_LSpdSetMotorCmd AND NOT #I_LSpdResMotorCmd AND NOT #I_HSpdSetMotorCmd AND NOT #I_HSpdResMotorCmd) OR (#I_LSpdResMotorCmd AND NOT #I_LSpdSetMotorCmd AND NOT #I_HSpdSetMotorCmd AND NOT #I_HSpdResMotorCmd) OR (#I_HSpdSetMotorCmd AND NOT #I_LSpdSetMotorCmd AND NOT #I_LSpdResMotorCmd AND NOT #I_HSpdResMotorCmd) OR (#I_HSpdResMotorCmd AND NOT #I_LSpdSetMotorCmd AND NOT #I_LSpdResMotorCmd AND NOT #I_HSpdSetMotorCmd)) AND #SafetyOk AND NOT #AA_MotorProtector AND NOT #AA_SafetySwitch AND NOT #DriveFaultAlarm;
   #Start := #_w1;   // Only 1 of the 4 commands may be active or else there is no start commend, if there is no start command the setpoint for the drive is also 0%
   IF NOT #_w1 THEN #SetpointSpeed := 0.0; END_IF;
END_REGION

REGION Network 27: **** 7.3 - Submodule - Machine **** MoviFit FC
   IF "TRUE" THEN
       #_MoviFitPN(I_ContolInhibit := "FALSE",   // "LGBSEW-MoviFitFCPN": Copy data with HW ID _________ /________ / l input telegram l SEW l l ===============>> PLC l Drive _l / <<=============== -l__l output telegram ********************************************************** SEW drive config: - 8.. Unit functions l - 87 Process data assignment _____________________ 870 Setpoint description PO1 l Control word 2 v l _____________________ 871 Setpoint description PO2 l Setpoint speed [%] v l _____________________ 872 Setpoint description PO3 l Ramp v l _____________________ 873 Actual value description PI1 l Status word 1 v l _____________________ 874 Actual value description PI2 l Output current v l _____________________ 875 Actual value description PI3 l Status word 2 v l _____________________ 876 PO data enable l Yes v l l v This changes to no when a POx paramater is changed Dot not forget to put this back to yes ! ********************************************************** "I_Ramp" is send to the drive in ms. Speed The ramp up / down time is (Rpm) ^ / set with this parameter l _________ / l / \/ l / \ l____/ \____ l--------------------------------------------------> t (s) _ ********************************************************** "I_OFF1" & "I_OFF2" example: ^ Speed (%) Stop signal at 5s l / 100% l______________/_ l \ \ l \ \ l \ \ l \ \ 0% l___________________\_____\___________________________> Time (s) l OFF2 OFF1 (regular start stop) 7s 10s Ramp down time settings to be done in the drive. OFF2 is to be used for controlled stops when there is a need to stop faster then regular, for example when there is an E-stop at a lift it is better to do a controlled stop and after that (x time in safety program) to give a STO. Note if there is a safe stop availible on safety level this is to be used instead of the non safety signals. _
                   I_OFF1 := #Start,
                   I_OFF2 := #C_Config.NotQuickStop,
                   I_ResetFault := #I_AlarmResetPB,
                   I_BrakeRelease := #I_ReleaseBrake AND #C_Config.ReleaseBrakeUsed,
                   I_ParameterSet := "FALSE",
                   I_SetpointSpeed := #SetpointSpeed,
                   I_Ramp := #RampToDrive,
                   C_HWSubInput := #C_Config.HWSubInput,
                   C_HWSubInputStatus := #C_Config.HWSubInputStatus,
                   C_HWSubOutput := #C_Config.HWSubOutput,
                   C_DriveCurrent := #C_Config.ReferenceDriveCurrent,
                   C_MotorCurrent := #C_Config.ReferenceMotorCurrent,
                   O_DriveReady => #DriveReady,
                   O_OutputStageEnabled => #OutputStageEnabled,
                   O_MaintenanceSwitch => #MaintenanceSwitch,
                   O_ParameterSet => #ParameterSet,
                   O_PODataEnabled => #PODataEnabled,
                   O_Fault => #Fault,
                   O_Brake => #Brake,
                   O_ActorVoltageOverloadDO00 => #ActorVoltageOverloadDO00,
                   O_ActorVoltageOverloadDO01 => #ActorVoltageOverloadDO01,
                   O_ActorVoltageOverloadDO02 => #ActorVoltageOverloadDO02,
                   O_ActorVoltageOverloadDO03 => #ActorVoltageOverloadDO03,
                   O_SensorVoltageOverloadGroup1 => #SensorVoltageOverloadGroup1,
                   O_SensorVoltageOverloadGroup2 => #SensorVoltageOverloadGroup2,
                   O_SensorVoltageOverloadGroup3 => #SensorVoltageOverloadGroup3,
                   O_SensorVoltageOverloadGroup4 => #SensorVoltageOverloadGroup4,
                   "O_Undervoltage24V-S" => #"Undervoltage24V-S",
                   "O_InverterVoltageNotApplied24V-P" => #"InverterVoltageNotApplied24V-P",
                   O_MOVIFITSystemFault => #MOVIFITSystemFault,
                   H_StatusWord1 => #"H_GBExtCross2W2S-MoviFitFCPN".H_StatusWord1[1].H_Word,
                   H_StatusWord2 => #"H_GBExtCross2W2S-MoviFitFCPN".H_StatusWord2[1].H_Word,
                   H_StatusWord3 => #"H_GBExtCross2W2S-MoviFitFCPN".H_StatusWord3[1].H_Word,
                   H_ControlWord => #"H_GBExtCross2W2S-MoviFitFCPN".H_ControlWord[1].H_Word,
                   H_SetpointSpeed => #"H_GBExtCross2W2S-MoviFitFCPN".H_SetpointSpeed[1].H_Word,
                   H_SetpointSpeedProCent => #"H_GBExtCross2W2S-MoviFitFCPN".H_SetpointSpeedProCent[1].H_Real,
                   H_SetpointRamp => "NotUsedInt",
                   H_ActualCurrentA => #"H_GBExtCross2W2S-MoviFitFCPN".H_ActualCurrentA[1].H_Real,
                   H_ActualCurrentProCent => #"H_GBExtCross2W2S-MoviFitFCPN".H_ActualCurrentProCent[1].H_Real,
                   H_ActualWarning => #"H_GBExtCross2W2S-MoviFitFCPN".H_ActualWarning[1].H_Int,
                   H_ActualFault => #"H_GBExtCross2W2S-MoviFitFCPN".H_ActualFault[1].H_Int);
   END_IF;
END_REGION

REGION Network 28: **** 8 - Outputs **** Brake
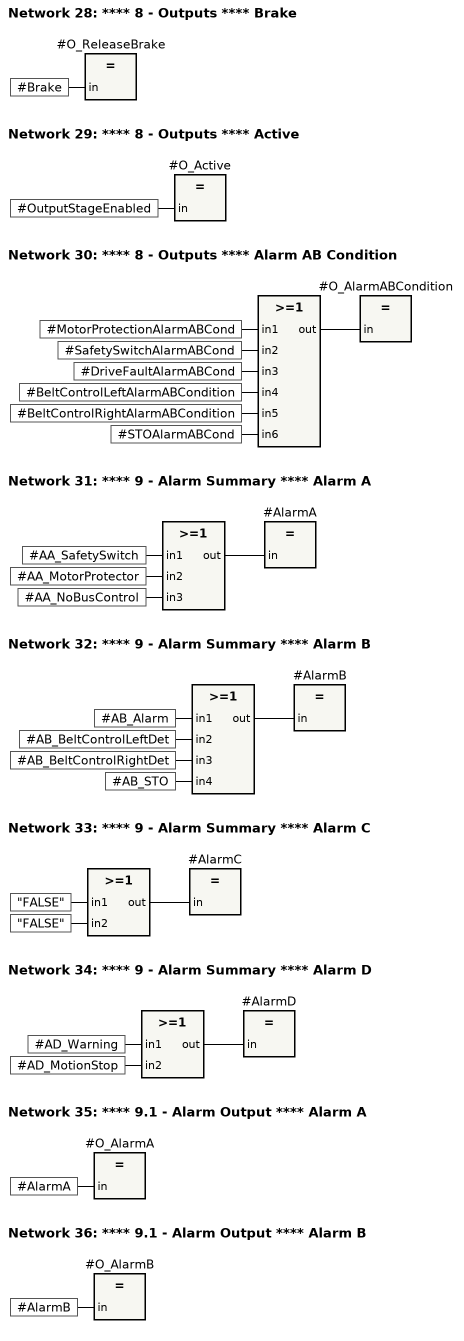
   #O_ReleaseBrake := #Brake;
END_REGION

REGION Network 29: **** 8 - Outputs **** Active
   // Active
   #O_Active := #OutputStageEnabled;
END_REGION

REGION Network 30: **** 8 - Outputs **** Alarm AB Condition
   // Alarm AB Condition
   #O_AlarmABCondition := #MotorProtectionAlarmABCond OR #SafetySwitchAlarmABCond OR #DriveFaultAlarmABCond OR #BeltControlLeftAlarmABCondition OR #BeltControlRightAlarmABCondition OR #STOAlarmABCond;
END_REGION

REGION Network 31: **** 9 - Alarm Summary **** Alarm A
   // Alarm A
   #AlarmA := #AA_SafetySwitch OR #AA_MotorProtector OR #AA_NoBusControl;
END_REGION

REGION Network 32: **** 9 - Alarm Summary **** Alarm B
   // Alarm B
   #AlarmB := #AB_Alarm OR #AB_BeltControlLeftDet OR #AB_BeltControlRightDet OR #AB_STO;
END_REGION

REGION Network 33: **** 9 - Alarm Summary **** Alarm C
   // Alarm C
   #AlarmC := "FALSE" OR "FALSE";
END_REGION

REGION Network 34: **** 9 - Alarm Summary **** Alarm D
   // Alarm D
   #AlarmD := #AD_Warning OR #AD_MotionStop;
END_REGION

REGION Network 35: **** 9.1 - Alarm Output **** Alarm A
   // Alarm A
   #O_AlarmA := #AlarmA;
END_REGION

REGION Network 36: **** 9.1 - Alarm Output **** Alarm B
   // Alarm B
   #O_AlarmB := #AlarmB;
END_REGION

REGION Network 37: **** 9.1 - Alarm Output **** Alarm C
   // Alarm C
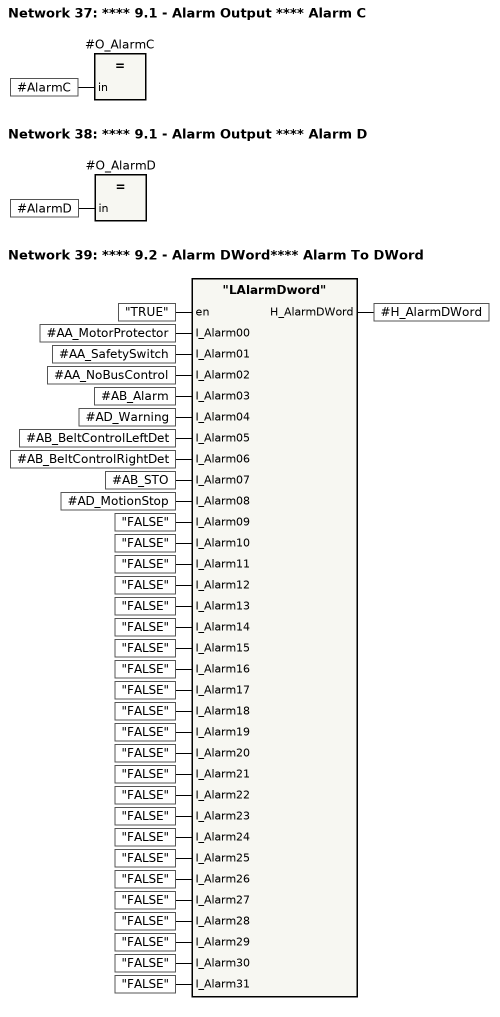
   #O_AlarmC := #AlarmC;
END_REGION

REGION Network 38: **** 9.1 - Alarm Output **** Alarm D
   // Alarm D
   #O_AlarmD := #AlarmD;
END_REGION

REGION Network 39: **** 9.2 - Alarm DWord**** Alarm To DWord
   // Alarm To Word
   IF "TRUE" THEN
       "LAlarmDword"(I_Alarm00 := #AA_MotorProtector,
                     I_Alarm01 := #AA_SafetySwitch,
                     I_Alarm02 := #AA_NoBusControl,
                     I_Alarm03 := #AB_Alarm,
                     I_Alarm04 := #AD_Warning,
                     I_Alarm05 := #AB_BeltControlLeftDet,
                     I_Alarm06 := #AB_BeltControlRightDet,
                     I_Alarm07 := #AB_STO,
                     I_Alarm08 := #AD_MotionStop,
                     I_Alarm09 := "FALSE",
                     I_Alarm10 := "FALSE",
                     I_Alarm11 := "FALSE",
                     I_Alarm12 := "FALSE",
                     I_Alarm13 := "FALSE",
                     I_Alarm14 := "FALSE",
                     I_Alarm15 := "FALSE",
                     I_Alarm16 := "FALSE",
                     I_Alarm17 := "FALSE",
                     I_Alarm18 := "FALSE",
                     I_Alarm19 := "FALSE",
                     I_Alarm20 := "FALSE",
                     I_Alarm21 := "FALSE",
                     I_Alarm22 := "FALSE",
                     I_Alarm23 := "FALSE",
                     I_Alarm24 := "FALSE",
                     I_Alarm25 := "FALSE",
                     I_Alarm26 := "FALSE",
                     I_Alarm27 := "FALSE",
                     I_Alarm28 := "FALSE",
                     I_Alarm29 := "FALSE",
                     I_Alarm30 := "FALSE",
                     I_Alarm31 := "FALSE",
                     H_AlarmDWord => #H_AlarmDWord);
   END_IF;
END_REGION
END_FUNCTION_BLOCK
